FUNCTION_BLOCK FB_PI
VAR_INPUT
	ssMethodType: SINT;
	fErr: LREAL;
	fP: LREAL;
	fI: LREAL;
END_VAR
VAR_OUTPUT
	fOut: LREAL;
END_VAR
VAR
	Integrator_DSTATE: LREAL;
END_VAR

CASE ssMethodType OF
    SS_INITIALIZE:         
        Integrator_DSTATE := 0.0;
    SS_STEP:       
        fOut := (fErr * fP) + Integrator_DSTATE;        
        Integrator_DSTATE := ((fErr * fI) * 0.01) + Integrator_DSTATE;
END_CASE;

END_FUNCTION_BLOCK

(* stored: Version 1.1.0.1, ProductVersion 3.1.4024.4
   POU FB_PI: Id {0aa1776b-29e4-45c6-9c54-b668de9c997d}, SpecialFunc None *)
